FUNCTION_BLOCK StackControl2
  (* Standard: 61499-2 *)
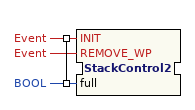
  EVENT_INPUT
    INIT WITH full;
    REMOVE_WP;
  END_EVENT
  VAR_INPUT
    full : BOOL;
  END_VAR
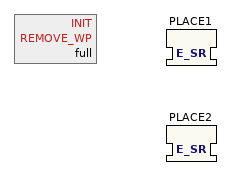
  FBS
    PLACE1 : E_SR;
    PLACE2 : E_SR;
  END_FBS
END_FUNCTION_BLOCK
